PROGRAM MAIN
VAR
END_VAR

END_PROGRAM

(* stored: Version 1.1.0.1
   POU MAIN: Id {3bae5e50-c07d-412a-938b-5e9efd473388} *)
